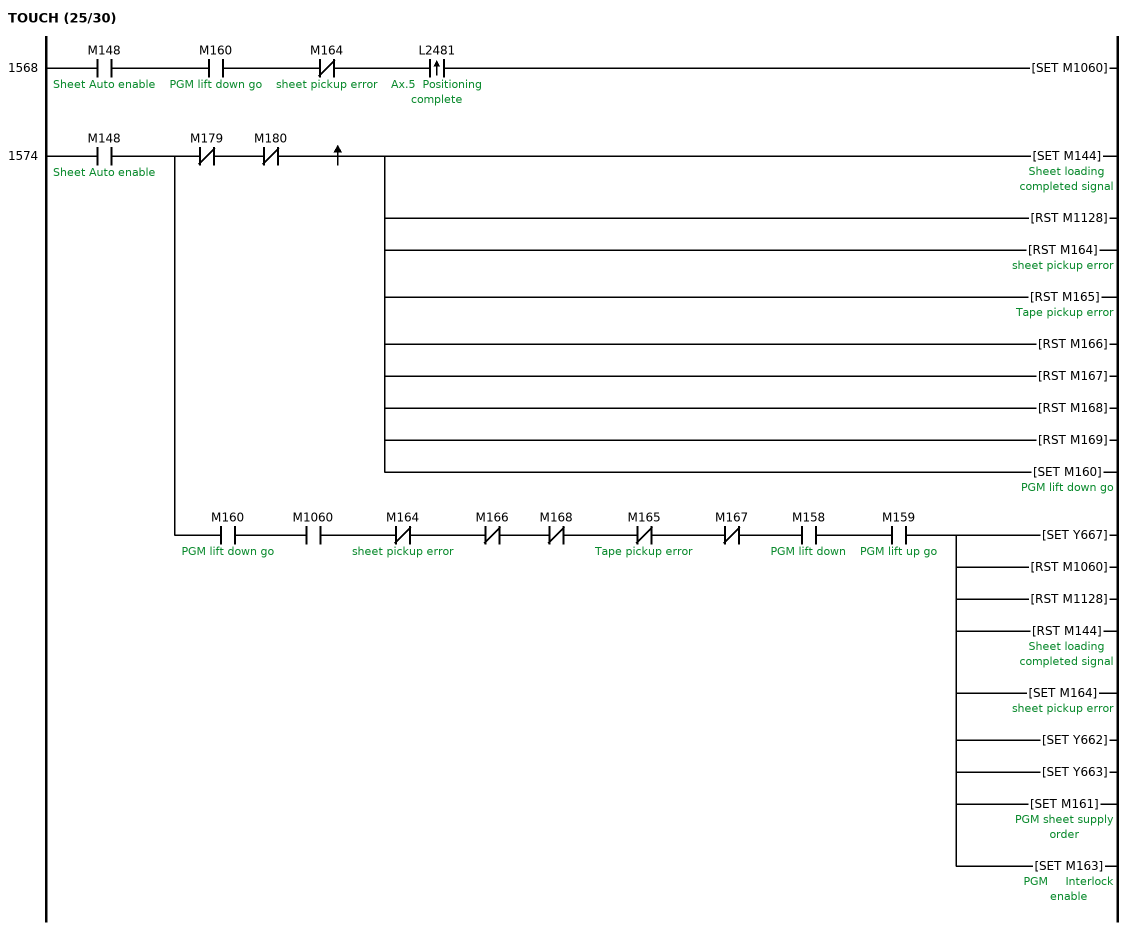
[picture p72: ladder of TOUCH, rungs at steps 1568 to 1574]
1568  LD      M148  ; Sheet Auto enable
      AND     M160  ; PGM lift down go
      ANI     M164  ; sheet pickup error
      ANDP    L2481  ; Ax.5  Positioning complete
      SET     M1060
1574  LD      M148  ; Sheet Auto enable
      MPS
      ANI     M179
      ANI     M180
      MEP
      SET     M144  ; Sheet loading completed signal
      RST     M1128
      RST     M164  ; sheet pickup error
      RST     M165  ; Tape pickup error
      RST     M166
      RST     M167
      RST     M168
      RST     M169
      SET     M160  ; PGM lift down go
      MPP
      AND     M160  ; PGM lift down go
      AND     M1060
      ANI     M164  ; sheet pickup error
      ANI     M166
      ANI     M168
      ANI     M165  ; Tape pickup error
      ANI     M167
      AND     M158  ; PGM lift down
      AND     M159  ; PGM lift up go
      SET     Y667
      RST     M1060
      RST     M1128
      RST     M144  ; Sheet loading completed signal
      SET     M164  ; sheet pickup error
      SET     Y662
      SET     Y663
      SET     M161  ; PGM sheet supply order
      SET     M163  ; PGM     Interlock enable
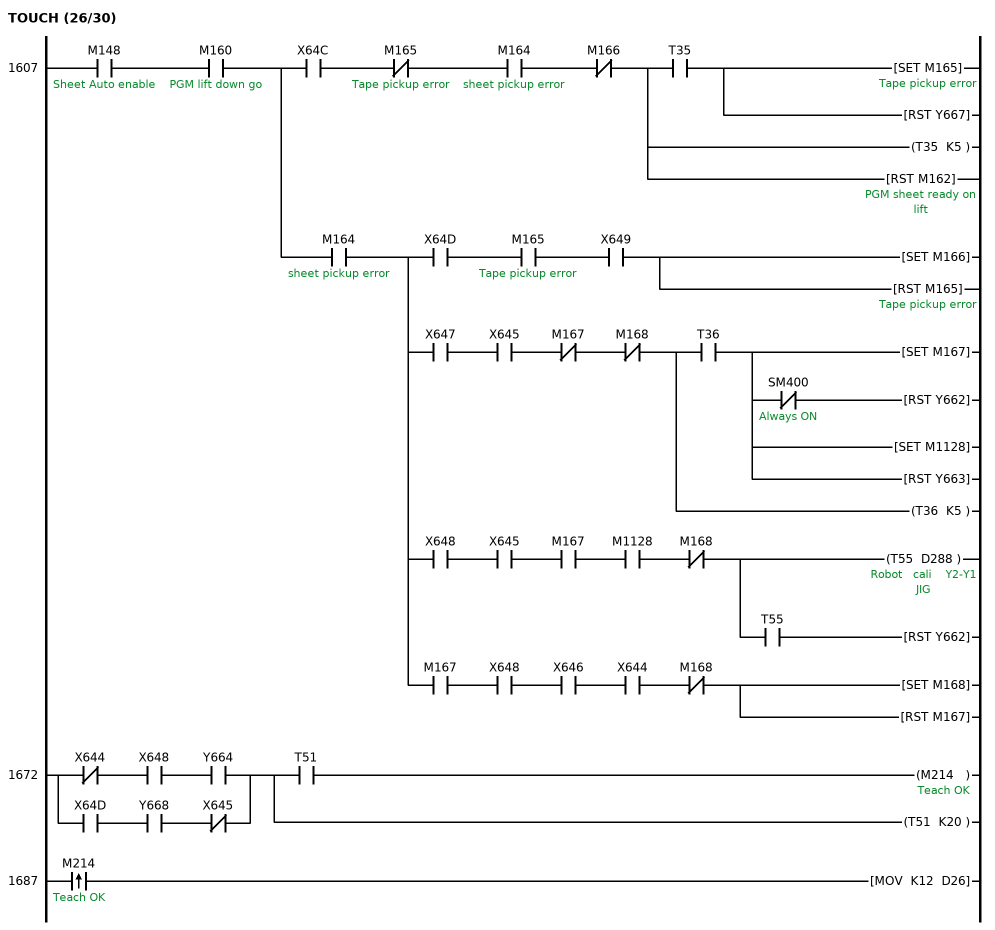
1607  LD      M148  ; Sheet Auto enable
      AND     M160  ; PGM lift down go
      MPS
      AND     X64C
      ANI     M165  ; Tape pickup error
      AND     M164  ; sheet pickup error
      ANI     M166
      MPS
      AND     T35
      SET     M165  ; Tape pickup error
      RST     Y667
      MPP
      OUT     T35 K5
      RST     M162  ; PGM sheet ready on lift
      MPP
      AND     M164  ; sheet pickup error
      MPS
      AND     X64D
      AND     M165  ; Tape pickup error
      AND     X649
      SET     M166
      RST     M165  ; Tape pickup error
      MRD
      AND     X647
      AND     X645
      ANI     M167
      ANI     M168
      MPS
      AND     T36
      SET     M167
      MPS
      ANI     SM400  ; Always ON
      RST     Y662
      MPP
      SET     M1128
      RST     Y663
      MPP
      OUT     T36 K5
      MRD
      AND     X648
      AND     X645
      AND     M167
      AND     M1128
      ANI     M168
      OUT     T55 D288  ; Robot   cali    Y2-Y1   JIG
      AND     T55
      RST     Y662
      MPP
      AND     M167
      AND     X648
      AND     X646
      AND     X644
      ANI     M168
      SET     M168
      RST     M167
1672  LDI     X644
      AND     X648
      AND     Y664
      LD      X64D
      AND     Y668
      ANI     X645
      ORB
      MPS
      AND     T51
      OUT     M214  ; Teach OK
      MPP
      OUT     T51 K20
1687  LDP     M214  ; Teach OK
      MOV     K12 D26
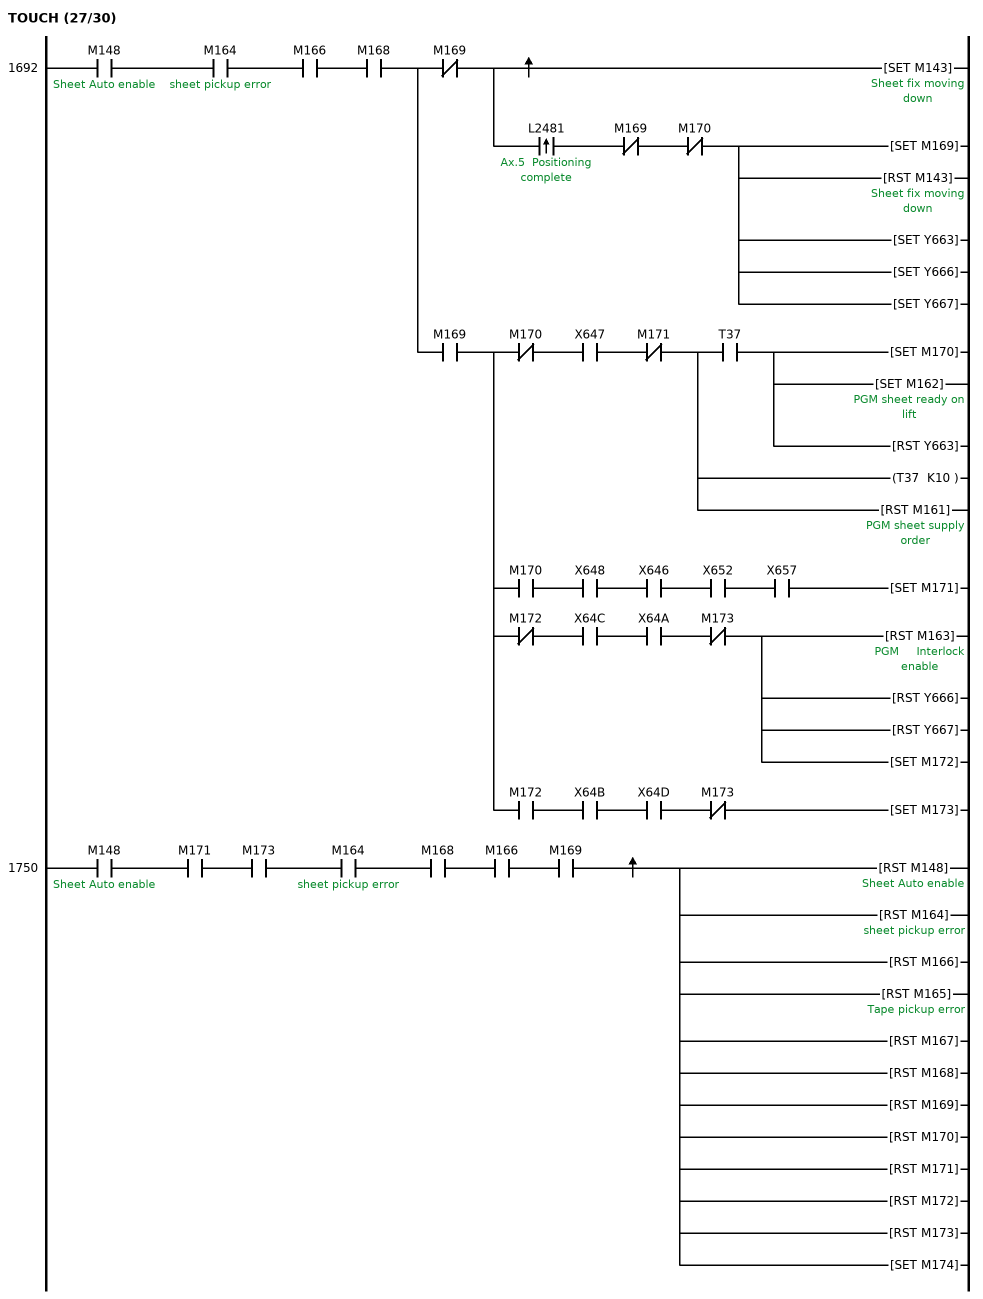
1692  LD      M148  ; Sheet Auto enable
      AND     M164  ; sheet pickup error
      AND     M166
      AND     M168
      MPS
      ANI     M169
      MPS
      MEP
      SET     M143  ; Sheet fix moving down
      MPP
      ANDP    L2481  ; Ax.5  Positioning complete
      ANI     M169
      ANI     M170
      SET     M169
      RST     M143  ; Sheet fix moving down
      SET     Y663
      SET     Y666
      SET     Y667
      MPP
      AND     M169
      MPS
      ANI     M170
      AND     X647
      ANI     M171
      MPS
      AND     T37
      SET     M170
      SET     M162  ; PGM sheet ready on lift
      RST     Y663
      MPP
      OUT     T37 K10
      RST     M161  ; PGM sheet supply order
      MRD
      AND     M170
      AND     X648
      AND     X646
      AND     X652
      AND     X657
      SET     M171
      MRD
      ANI     M172
      AND     X64C
      AND     X64A
      ANI     M173
      RST     M163  ; PGM     Interlock enable
      RST     Y666
      RST     Y667
      SET     M172
      MPP
      AND     M172
      AND     X64B
      AND     X64D
      ANI     M173
      SET     M173
1750  LD      M148  ; Sheet Auto enable
      AND     M171
      AND     M173
      AND     M164  ; sheet pickup error
      AND     M168
      AND     M166
      AND     M169
      MEP
      RST     M148  ; Sheet Auto enable
      RST     M164  ; sheet pickup error
      RST     M166
      RST     M165  ; Tape pickup error
      RST     M167
      RST     M168
      RST     M169
      RST     M170
      RST     M171
      RST     M172
      RST     M173
      SET     M174
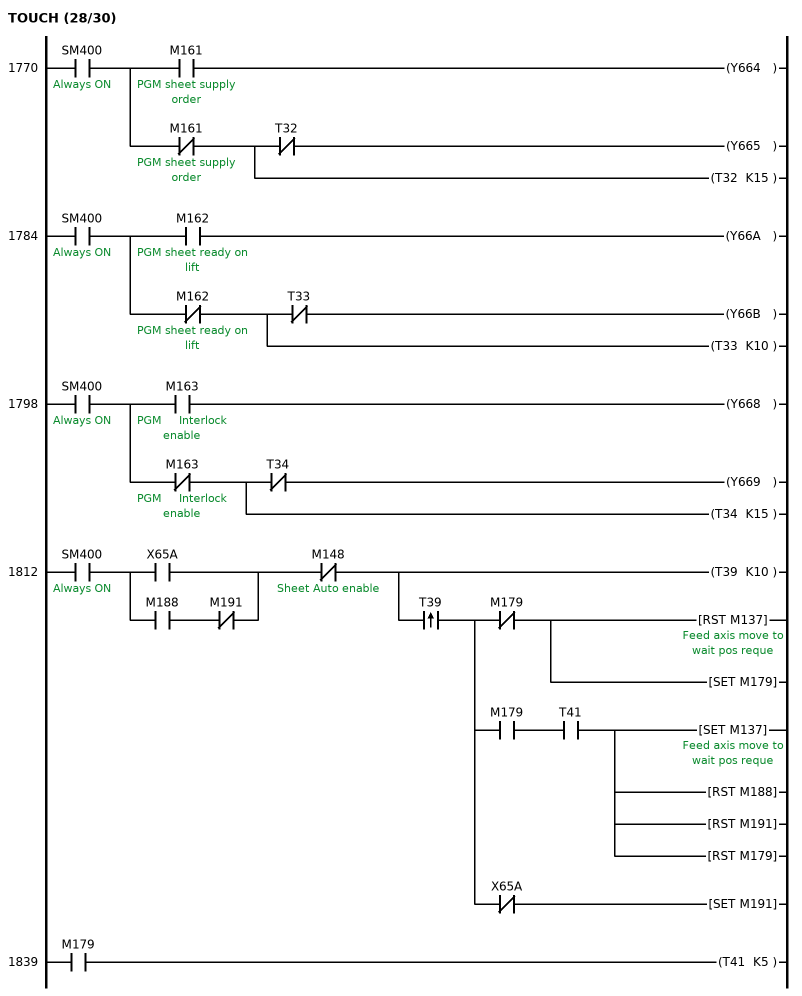
1770  LD      SM400  ; Always ON
      MPS
      AND     M161  ; PGM sheet supply order
      OUT     Y664
      MPP
      ANI     M161  ; PGM sheet supply order
      MPS
      ANI     T32
      OUT     Y665
      MPP
      OUT     T32 K15
1784  LD      SM400  ; Always ON
      MPS
      AND     M162  ; PGM sheet ready on lift
      OUT     Y66A
      MPP
      ANI     M162  ; PGM sheet ready on lift
      MPS
      ANI     T33
      OUT     Y66B
      MPP
      OUT     T33 K10
1798  LD      SM400  ; Always ON
      MPS
      AND     M163  ; PGM     Interlock enable
      OUT     Y668
      MPP
      ANI     M163  ; PGM     Interlock enable
      MPS
      ANI     T34
      OUT     Y669
      MPP
      OUT     T34 K15
1812  LD      SM400  ; Always ON
      LD      X65A
      LD      M188
      ANI     M191
      ORB
      ANB
      ANI     M148  ; Sheet Auto enable
      OUT     T39 K10
      ANDP    T39
      MPS
      ANI     M179
      RST     M137  ; Feed axis move to wait pos reque
      SET     M179
      MRD
      AND     M179
      AND     T41
      SET     M137  ; Feed axis move to wait pos reque
      RST     M188
      RST     M191
      RST     M179
      MPP
      ANI     X65A
      SET     M191
1839  LD      M179
      OUT     T41 K5
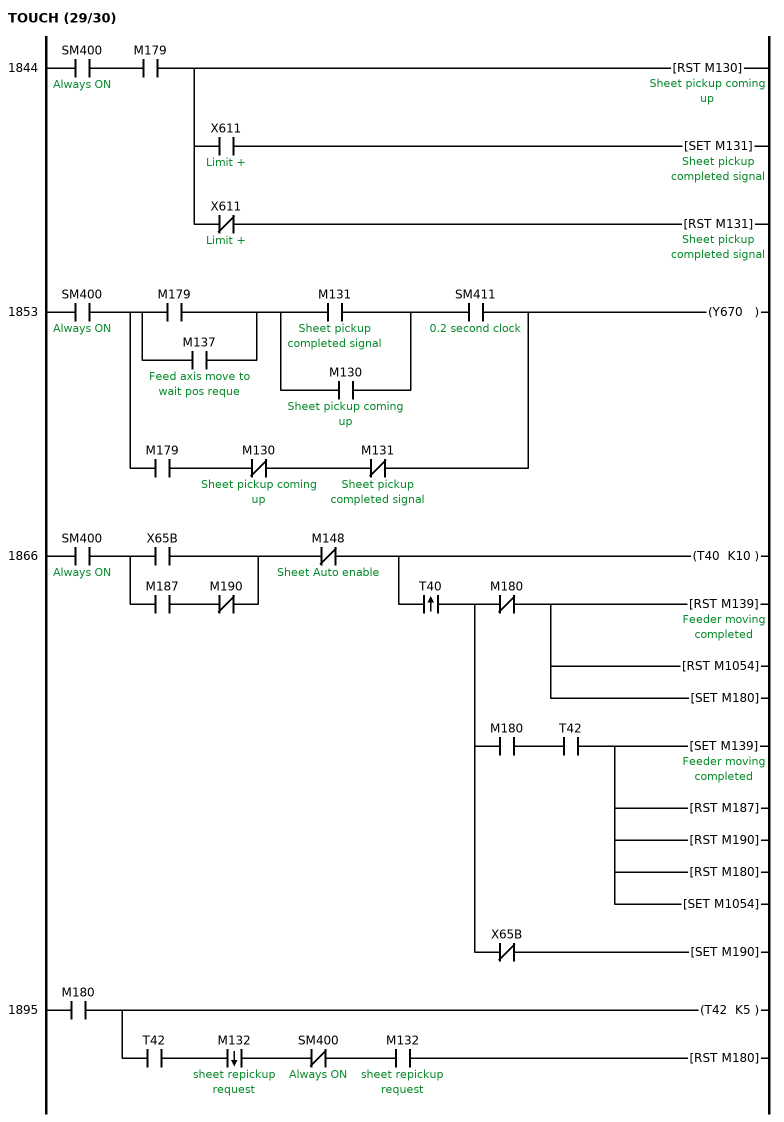
1844  LD      SM400  ; Always ON
      AND     M179
      RST     M130  ; Sheet pickup coming up
      MPS
      AND     X611  ; Limit +
      SET     M131  ; Sheet pickup completed signal
      MPP
      ANI     X611  ; Limit +
      RST     M131  ; Sheet pickup completed signal
1853  LD      SM400  ; Always ON
      LD      M179
      OR      M137  ; Feed axis move to wait pos reque
      LD      M131  ; Sheet pickup completed signal
      OR      M130  ; Sheet pickup coming up
      ANB
      AND     SM411  ; 0.2 second clock
      LD      M179
      ANI     M130  ; Sheet pickup coming up
      ANI     M131  ; Sheet pickup completed signal
      ORB
      ANB
      OUT     Y670
1866  LD      SM400  ; Always ON
      LD      X65B
      LD      M187
      ANI     M190
      ORB
      ANB
      ANI     M148  ; Sheet Auto enable
      OUT     T40 K10
      ANDP    T40
      MPS
      ANI     M180
      RST     M139  ; Feeder moving completed
      RST     M1054
      SET     M180
      MRD
      AND     M180
      AND     T42
      SET     M139  ; Feeder moving completed
      RST     M187
      RST     M190
      RST     M180
      SET     M1054
      MPP
      ANI     X65B
      SET     M190
1895  LD      M180
      OUT     T42 K5
      AND     T42
      ANDF    M132  ; sheet repickup request
      ANI     SM400  ; Always ON
      AND     M132  ; sheet repickup request
      RST     M180
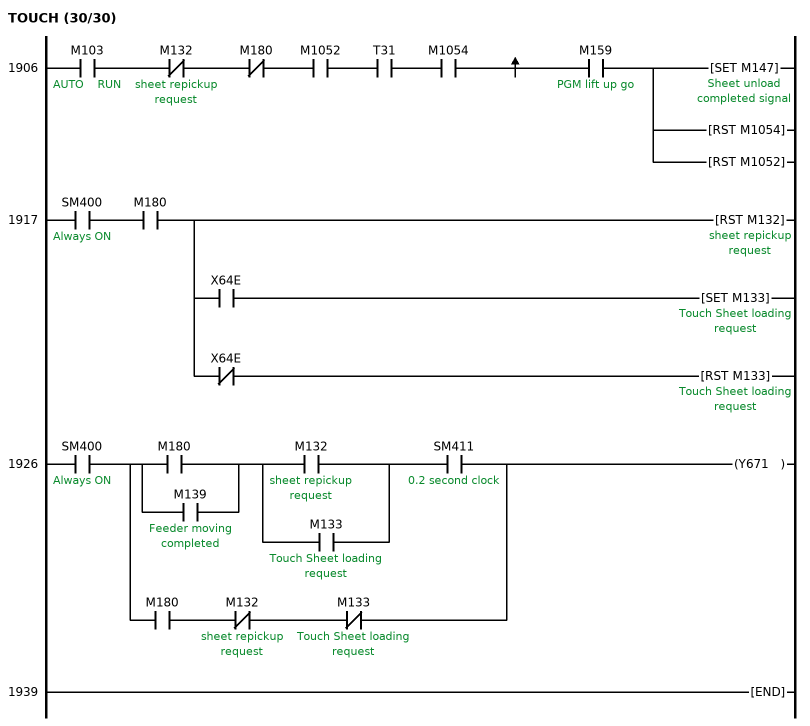
1906  LD      M103  ; AUTO    RUN
      ANI     M132  ; sheet repickup request
      ANI     M180
      AND     M1052
      AND     T31
      AND     M1054
      MEP
      AND     M159  ; PGM lift up go
      SET     M147  ; Sheet unload completed signal
      RST     M1054
      RST     M1052
1917  LD      SM400  ; Always ON
      AND     M180
      RST     M132  ; sheet repickup request
      MPS
      AND     X64E
      SET     M133  ; Touch Sheet loading request
      MPP
      ANI     X64E
      RST     M133  ; Touch Sheet loading request
1926  LD      SM400  ; Always ON
      LD      M180
      OR      M139  ; Feeder moving completed
      LD      M132  ; sheet repickup request
      OR      M133  ; Touch Sheet loading request
      ANB
      AND     SM411  ; 0.2 second clock
      LD      M180
      ANI     M132  ; sheet repickup request
      ANI     M133  ; Touch Sheet loading request
      ORB
      ANB
      OUT     Y671
1939  END
END_PROGRAM

PROGRAM VISION
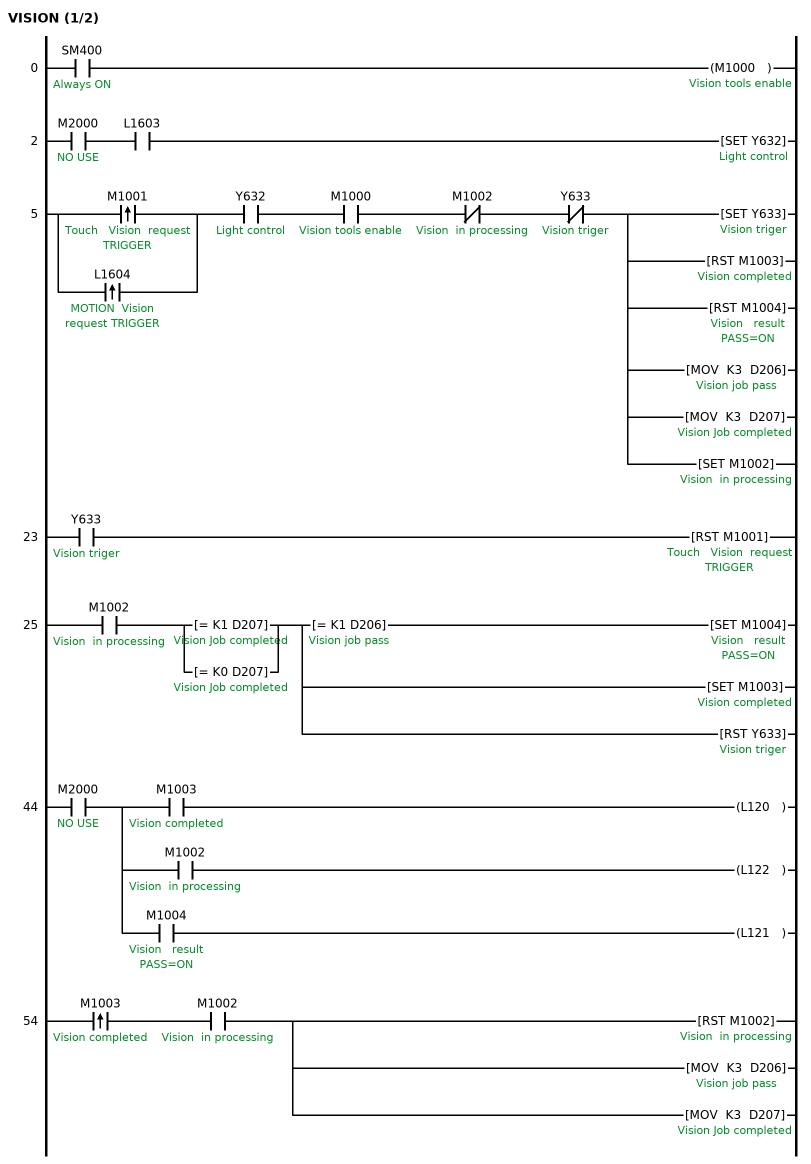
0     LD      SM400  ; Always ON
      OUT     M1000  ; Vision tools enable
2     LD      M2000  ; NO USE
      AND     L1603
      SET     Y632  ; Light control
5     LDP     M1001  ; Touch   Vision  request TRIGGER
      ORP     L1604  ; MOTION  Vision  request TRIGGER
      AND     Y632  ; Light control
      AND     M1000  ; Vision tools enable
      ANI     M1002  ; Vision  in processing
      ANI     Y633  ; Vision triger
      SET     Y633  ; Vision triger
      RST     M1003  ; Vision completed
      RST     M1004  ; Vision   result PASS=ON
      MOV     K3 D206  ; Vision job pass
      MOV     K3 D207  ; Vision Job completed
      SET     M1002  ; Vision  in processing
23    LD      Y633  ; Vision triger
      RST     M1001  ; Touch   Vision  request TRIGGER
25    LD      M1002  ; Vision  in processing
      LD=     K1 D207  ; Vision Job completed
      OR=     K0 D207  ; Vision Job completed
      ANB
      MPS
      AND=    K1 D206  ; Vision job pass
      SET     M1004  ; Vision   result PASS=ON
      MPP
      SET     M1003  ; Vision completed
      RST     Y633  ; Vision triger
44    LD      M2000  ; NO USE
      MPS
      AND     M1003  ; Vision completed
      OUT     L120
      MRD
      AND     M1002  ; Vision  in processing
      OUT     L122
      MPP
      AND     M1004  ; Vision   result PASS=ON
      OUT     L121
54    LDP     M1003  ; Vision completed
      AND     M1002  ; Vision  in processing
      RST     M1002  ; Vision  in processing
      MOV     K3 D206
      MOV     K3 D207
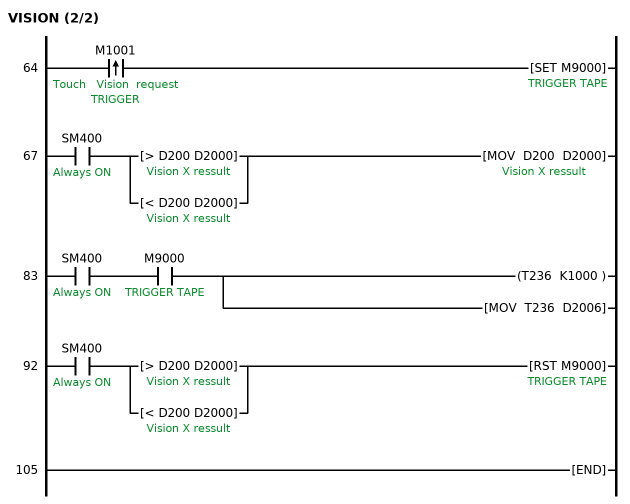
64    LDP     M1001  ; Touch   Vision  request TRIGGER
      SET     M9000  ; TRIGGER TAPE
67    LD      SM400  ; Always ON
      LD>     D200 D2000  ; Vision X ressult
      OR<     D200 D2000  ; Vision X ressult
      ANB
      MOV     D200 D2000
83    LD      SM400  ; Always ON
      AND     M9000  ; TRIGGER TAPE
      OUT     T236 K1000
      MOV     T236 D2006
92    LD      SM400  ; Always ON
      LD>     D200 D2000  ; Vision X ressult
      OR<     D200 D2000  ; Vision X ressult
      ANB
      RST     M9000  ; TRIGGER TAPE
105   END
END_PROGRAM

// device comments not shown above
X608  ; Vaccum pressure signal
X609  ; Change Tape
X61A  ; Fix sheet cylinder pos
X61E  ; Up Position
M10  ; Head Select
M30  ; Jig Vacuum-Blow
M219  ; CALIB OK
M220  ; CALIB   JIG OK
M270  ; SP_TRIG MCR
M300  ; nâng hạ bàn đặt Tape
M500  ; PROCESS PASS
M501  ; 1: DÁN 0: BỎ  QUA
M505  ; LUÔN   DÁN    TAPE
M1015  ; Vision  result  PASS=ON JIG1
M1024  ; Vision  result  PASS=ON JIG2
M1042  ; Get     vision  master  JIG
M1065  ; Robot   calib   Pos 1   get JIG
M1066  ; Robot   calib   Pos 2   get JIG
M1067  ; Robot   calib   excute  JIG
M1193  ; NO USE
D18  ; Sheet Rows
D20  ; Sheet rows index
D22  ; sheet repickup counter
D50  ; Vision X ressult JIG 1
D52  ; Vision Y result JIG 1
D54  ; Vision  angle JIG 1
D70  ; Vision X ressult JIG 2
D72  ; Vision Y result JIG 2
D74  ; Vision  angle JIG 2
D240  ; RB-CAM  RATE X  JIG
D242  ; RB-CAM  RATE Y  JIG
D250  ; Vision master X JIG1
D252  ; Vision master Y JIG1
D254  ; Vision master Angle JIG1
D260  ; Vision master X JIG2
D262  ; Vision master Y JIG2
D264  ; Vision master Angle JIG2
D270  ; Robot   cali X1 JIG
D272  ; Robot   cali Y1 JIG
D274  ; Robot   cali XC1 JIG
D276  ; Robot   cali YC1 JIG
D278  ; Robot   cali    X2-X1   JIG
D280  ; Robot   cali X2 JIG
D282  ; Robot   cali Y2 JIG
D286  ; Robot   cali YC2 JIG
D302  ; DO LECH YC JIG1
D304  ; GOCS2-  GÓC1   JIG1
D306  ; DO LECH XC JIG2
D308  ; DO LECH YC JIG2
D310  ; GOCS2-  GÓC1   JIG2    FLOAD
D312  ; BÙ XUNG XC JIG1
D314  ; BÙ XUNG YC JIG1
D316  ; BÙ XUNG XC JIG2
D318  ; BÙ XUNG YC JIG2
D320  ; INT BÙ XUNG JIG1 XC
D322  ; INT BÙ XUNG JIG1 YC
D380  ; VISION  HEAD 1  ANGLE
D382  ; VISION  HEAD 2  ANGLE
D48008  ; SPEED Z1 MANUAL
D48018  ; SPEED R1 MANUAL
D48028  ; SPEED Z2 MANUAL
D48038  ; SPEED R2 MANUAL
D48048  ; SPEED F MANUAL
D48050  ; ADRES X
D48052  ; SPEED X
D48058  ; SPEED X MANUAL
D48060  ; ADRES Y
D48062  ; SPEED Y
D48068  ; SPEED Y MANUAL
D48120  ; TIME    DELAY   RUN Z1, R1
D48640  ; Ax.1 JOG speed setting
D48641  ; Ax.1 JOG speed setting
D48642  ; Ax.2 JOG speed setting
D48643  ; Ax.2 JOG speed setting
D48644  ; Ax.3 JOG speed setting
D48645  ; Ax.3 JOG speed setting
D48646  ; Ax.4 JOG speed setting
D48647  ; Ax.4 JOG speed setting
D48648  ; Ax.5 JOG speed setting
D48649  ; Ax.5 JOG speed setting
D48650  ; Ax.6 JOG speed setting
D48651  ; Ax.6 JOG speed setting
D48652  ; Ax.7 JOG speed setting
D48653  ; Ax.7 JOG speed setting
D48654  ; Ax.8 JOG speed setting
D48655  ; Ax.8 JOG speed setting
D49000  ; Ax.1  Feed current value/Roller
D49001  ; Ax.1  Feed current value/Roller
D49003  ; Ax.1  Real current value
D49004  ; Ax.1  Deviation counter value
D49005  ; Ax.1  Deviation counter value
D49006  ; Ax.1  Minor error code
D49007  ; Ax.1  Major error code
D49008  ; Ax.1  Servo error code
D49009  ; Ax.1  Home position return re-mo
D49010  ; Ax.1  Movement amount after prox
D49011  ; Ax.1  Movement amount after prox
D49012  ; Ax.1  Execute program No.
D49013  ; Ax.1 M-code
D49014  ; Ax.1  Torque limit value
D49015  ; Ax.1  Data set pointer for const
D49018  ; Ax.1  Real current value at stop
D49019  ; Ax.1  Real current value at stop
D49020  ; Ax.2  Feed current value/Roller
D49021  ; Ax.2  Feed current value/Roller
D49023  ; Ax.2  Real current value
D49024  ; Ax.2  Deviation counter value
D49025  ; Ax.2  Deviation counter value
D49026  ; Ax.2  Minor error code
D49027  ; Ax.2  Major error code
D49028  ; Ax.2  Servo error code
D49029  ; Ax.2  Home position return re-mo
D49030  ; Ax.2  Movement amount after prox
D49031  ; Ax.2  Movement amount after prox
D49032  ; Ax.2  Execute program No.
D49033  ; Ax.2 M-code
D49034  ; Ax.2  Torque limit value
D49035  ; Ax.2  Data set pointer for const
D49038  ; Ax.2  Real current value at stop
D49039  ; Ax.2  Real current value at stop
D49040  ; Ax.3  Feed current value/Roller
D49041  ; Ax.3  Feed current value/Roller
D49043  ; Ax.3  Real current value
D49044  ; Ax.3  Deviation counter value
D49045  ; Ax.3  Deviation counter value
D49046  ; Ax.3  Minor error code
D49047  ; Ax.3  Major error code
D49048  ; Ax.3  Servo error code
D49049  ; Ax.3  Home position return re-mo
D49050  ; Ax.3  Movement amount after prox
D49051  ; Ax.3  Movement amount after prox
D49052  ; Ax.3  Execute program No.
D49053  ; Ax.3 M-code
D49054  ; Ax.3  Torque limit value
D49055  ; Ax.3  Data set pointer for const
D49058  ; Ax.3  Real current value at stop
D49059  ; Ax.3  Real current value at stop
D49060  ; Ax.4  Feed current value/Roller
D49061  ; Ax.4  Feed current value/Roller
D49063  ; Ax.4  Real current value
D49064  ; Ax.4  Deviation counter value
D49065  ; Ax.4  Deviation counter value
D49066  ; Ax.4  Minor error code
D49067  ; Ax.4  Major error code
D49068  ; Ax.4  Servo error code
D49069  ; Ax.4  Home position return re-mo
D49070  ; Ax.4  Movement amount after prox
D49071  ; Ax.4  Movement amount after prox
D49072  ; Ax.4  Execute program No.
D49073  ; Ax.4 M-code
D49074  ; Ax.4  Torque limit value
D49075  ; Ax.4  Data set pointer for const
D49078  ; Ax.4  Real current value at stop
D49079  ; Ax.4  Real current value at stop
D49080  ; Ax.5  Feed current value/Roller
D49081  ; Ax.5  Feed current value/Roller
D49083  ; Ax.5  Real current value
D49084  ; Ax.5  Deviation counter value
D49085  ; Ax.5  Deviation counter value
D49086  ; Ax.5  Minor error code
D49087  ; Ax.5  Major error code
D49088  ; Ax.5  Servo error code
D49089  ; Ax.5  Home position return re-mo
D49090  ; Ax.5  Movement amount after prox
D49091  ; Ax.5  Movement amount after prox
D49092  ; Ax.5  Execute program No.
D49093  ; Ax.5 M-code
D49094  ; Ax.5  Torque limit value
D49095  ; Ax.5  Data set pointer for const
D49098  ; Ax.5  Real current value at stop
D49099  ; Ax.5  Real current value at stop
D49100  ; Ax.6  Feed current value/Roller
D49101  ; Ax.6  Feed current value/Roller
D49103  ; Ax.6  Real current value
D49104  ; Ax.6  Deviation counter value
D49105  ; Ax.6  Deviation counter value
D49106  ; Ax.6  Minor error code
D49107  ; Ax.6  Major error code
D49108  ; Ax.6  Servo error code
D49109  ; Ax.6  Home position return re-mo
D49110  ; Ax.6  Movement amount after prox
D49111  ; Ax.6  Movement amount after prox
D49112  ; Ax.6  Execute program No.
D49113  ; Ax.6 M-code
D49114  ; Ax.6  Torque limit value
D49115  ; Ax.6  Data set pointer for const
D49118  ; Ax.6  Real current value at stop
D49119  ; Ax.6  Real current value at stop
D49120  ; Ax.7  Feed current value/Roller
D49121  ; Ax.7  Feed current value/Roller
D49123  ; Ax.7  Real current value
D49124  ; Ax.7  Deviation counter value
D49125  ; Ax.7  Deviation counter value
D49126  ; Ax.7  Minor error code
D49127  ; Ax.7  Major error code
D49128  ; Ax.7  Servo error code
D49129  ; Ax.7  Home position return re-mo
D49130  ; Ax.7  Movement amount after prox
D49131  ; Ax.7  Movement amount after prox
D49132  ; Ax.7  Execute program No.
D49133  ; Ax.7 M-code
D49134  ; Ax.7  Torque limit value
D49135  ; Ax.7  Data set pointer for const
D49138  ; Ax.7  Real current value at stop
D49139  ; Ax.7  Real current value at stop
D49140  ; Ax.8  Feed current value/Roller
D49141  ; Ax.8  Feed current value/Roller
D49142  ; Ax.8  Real current value
D49143  ; Ax.8  Real current value
D49144  ; Ax.8  Deviation counter value
D49145  ; Ax.8  Deviation counter value
D49146  ; Ax.8  Minor error code
D49147  ; Ax.8  Major error code
D49148  ; Ax.8  Servo error code
D49149  ; Ax.8  Home position return re-mo
D49150  ; Ax.8  Movement amount after prox
D49151  ; Ax.8  Movement amount after prox
D49152  ; Ax.8  Execute program No.
D49153  ; Ax.8 M-code
D49154  ; Ax.8  Torque limit value
D49155  ; Ax.8  Data set pointer for const
D49158  ; Ax.8  Real current value at stop
D49159  ; Ax.8  Real current value at stop
D49704  ; PLC ready flag request
D49705  ; Speed switching point specified
D49706  ; All axes servo ON command reques
D49714  ; Manual pulse generator 1 axis No
D49715  ; Manual pulse generator 1 axis No
D49716  ; Manual pulse generator 2 axis No
D49717  ; Manual pulse generator 2 axis No
D49718  ; Manual pulse generator 3 axis No
D49719  ; Manual pulse generator 3 axis No
D49720  ; Ax.1  ManualPulseGen. 1Pls. inpu
D49721  ; Ax.2  ManualPulseGen. 1Pls. inpu
D49722  ; Ax.3  ManualPulseGen. 1Pls. inpu
D49723  ; Ax.4  ManualPulseGen. 1Pls. inpu
D49724  ; Ax.5  ManualPulseGen. 1Pls. inpu
D49725  ; Ax.6  ManualPulseGen. 1Pls. inpu
D49726  ; Ax.7  ManualPulseGen. 1Pls. inpu
D49727  ; Ax.8  ManualPulseGen. 1Pls. inpu
D49752  ; Manual pulse generator 1 smoothi
D49753  ; Manual pulse generator 2 smoothi
D49754  ; Manual pulse generator 3 smoothi
D49755  ; Manual pulse generator 1 enable
D49756  ; Manual pulse generator 2 enable
D49757  ; Manual pulse generator 3 enable
D49800  ; Virtual servo  Ax.1  Feed curren
D49801  ; Virtual servo  Ax.1  Feed curren
D49802  ; Virtual servo  Ax.1  Minor error
D49803  ; Virtual servo  Ax.1  Major error
D49804  ; Virtual servo  Ax.1  Execute pro
D49805  ; Virtual servo  Ax.1  M-code
D49806  ; Virtual servo  Ax.1  Current val
D49807  ; Virtual servo  Ax.1  Current val
D49808  ; Virtual servo  Ax.1  Error searc
D49809  ; Virtual servo  Ax.1  Data set po
D49810  ; Virtual servo  Ax.2  Feed curren
D49811  ; Virtual servo  Ax.2  Feed curren
D49812  ; Virtual servo  Ax.2  Minor error
D49813  ; Virtual servo  Ax.2  Major error
D49814  ; Virtual servo  Ax.2  Execute pro
D49815  ; Virtual servo  Ax.2  M-code
D49816  ; Virtual servo  Ax.2  Current val
D49817  ; Virtual servo  Ax.2  Current val
D49818  ; Virtual servo  Ax.2  Error searc
D49819  ; Virtual servo  Ax.2  Data set po
D49820  ; Virtual servo  Ax.3  Feed curren
D49821  ; Virtual servo  Ax.3  Feed curren
D49822  ; Virtual servo  Ax.3  Minor error
D49823  ; Virtual servo  Ax.3  Major error
D49824  ; Virtual servo  Ax.3  Execute pro
D49825  ; Virtual servo  Ax.3  M-code
D49826  ; Virtual servo  Ax.3  Current val
D49827  ; Virtual servo  Ax.3  Current val
D49828  ; Virtual servo  Ax.3  Error searc
D49829  ; Virtual servo  Ax.3  Data set po
D49830  ; Virtual servo  Ax.4  Feed curren
D49831  ; Virtual servo  Ax.4  Feed curren
D49832  ; Virtual servo  Ax.4  Minor error
D49833  ; Virtual servo  Ax.4  Major error
D49834  ; Virtual servo  Ax.4  Execute pro
D49835  ; Virtual servo  Ax.4  M-code
D49836  ; Virtual servo  Ax.4  Current val
D49837  ; Virtual servo  Ax.4  Current val
D49838  ; Virtual servo  Ax.4  Error searc
D49839  ; Virtual servo  Ax.4  Data set po
D49840  ; Virtual servo  Ax.5  Feed curren
D49841  ; Virtual servo  Ax.5  Feed curren
D49842  ; Virtual servo  Ax.5  Minor error
D49843  ; Virtual servo  Ax.5  Major error
D49844  ; Virtual servo  Ax.5  Execute pro
D49845  ; Virtual servo  Ax.5  M-code
D49846  ; Virtual servo  Ax.5  Current val
D49847  ; Virtual servo  Ax.5  Current val
D49848  ; Virtual servo  Ax.5  Error searc
D49849  ; Virtual servo  Ax.5  Data set po
D49850  ; Virtual servo  Ax.6  Feed curren
D49851  ; Virtual servo  Ax.6  Feed curren
D49852  ; Virtual servo  Ax.6  Minor error
D49853  ; Virtual servo  Ax.6  Major error
D49854  ; Virtual servo  Ax.6  Execute pro
D49855  ; Virtual servo  Ax.6  M-code
D49856  ; Virtual servo  Ax.6  Current val
D49857  ; Virtual servo  Ax.6  Current val
D49858  ; Virtual servo  Ax.6  Error searc
D49859  ; Virtual servo  Ax.6  Data set po
D49860  ; Virtual servo  Ax.7  Feed curren
D49861  ; Virtual servo  Ax.7  Feed curren
D49862  ; Virtual servo  Ax.7  Minor error
D49863  ; Virtual servo  Ax.7  Major error
D49864  ; Virtual servo  Ax.7  Execute pro
D49865  ; Virtual servo  Ax.7  M-code
D49866  ; Virtual servo  Ax.7  Current val
D49867  ; Virtual servo  Ax.7  Current val
D49868  ; Virtual servo  Ax.7  Error searc
D49869  ; Virtual servo  Ax.7  Data set po
D49870  ; Virtual servo  Ax.8  Feed curren
D49871  ; Virtual servo  Ax.8  Feed curren
D49872  ; Virtual servo  Ax.8  Minor error
D49873  ; Virtual servo  Ax.8  Major error
D49874  ; Virtual servo  Ax.8  Execute pro
D49875  ; Virtual servo  Ax.8  M-code
D49876  ; Virtual servo  Ax.8  Current val
D49877  ; Virtual servo  Ax.8  Current val
D49878  ; Virtual servo  Ax.8  Error searc
D49879  ; Virtual servo  Ax.8  Data set po
D50122  ; Sync. encoder  Ax.1  Minor error
D50123  ; Sync. encoder  Ax.1  Major error
D50128  ; Sync. encoder  Ax.1  Error searc
D50132  ; Sync. encoder  Ax.2  Minor error
D50133  ; Sync. encoder  Ax.2  Major error
D50138  ; Sync. encoder  Ax.2  Error searc
D50142  ; Sync. encoder  Ax.3  Minor error
D50143  ; Sync. encoder  Ax.3  Major error
D50148  ; Sync. encoder  Ax.3  Error searc
D50152  ; Sync. encoder  Ax.4  Minor error
D50153  ; Sync. encoder  Ax.4  Major error
D50158  ; Sync. encoder  Ax.4  Error searc
D50162  ; Sync. encoder  Ax.5  Minor error
D50163  ; Sync. encoder  Ax.5  Major error
D50168  ; Sync. encoder  Ax.5  Error searc
D50172  ; Sync. encoder  Ax.6  Minor error
D50173  ; Sync. encoder  Ax.6  Major error
D50178  ; Sync. encoder  Ax.6  Error searc
D50182  ; Sync. encoder  Ax.7  Minor error
D50183  ; Sync. encoder  Ax.7  Major error
D50188  ; Sync. encoder  Ax.7  Error searc
D50192  ; Sync. encoder  Ax.8  Minor error
D50193  ; Sync. encoder  Ax.8  Major error
D50198  ; Sync. encoder  Ax.8  Error searc
D50241  ; Cam  Ax.1  Execute cam No.
D50242  ; Cam  Ax.1  Execute stroke amount
D50243  ; Cam  Ax.1  Execute stroke amount
D50244  ; Cam  Ax.1  Cam axis current valu
D50245  ; Cam  Ax.1  Cam axis current valu
D50251  ; Cam  Ax.2  Execute cam No.
D50252  ; Cam  Ax.2  Execute stroke amount
D50253  ; Cam  Ax.2  Execute stroke amount
D50254  ; Cam  Ax.2  Cam axis current valu
D50255  ; Cam  Ax.2  Cam axis current valu
D50261  ; Cam  Ax.3  Execute cam No.
D50262  ; Cam  Ax.3  Execute stroke amount
D50263  ; Cam  Ax.3  Execute stroke amount
D50264  ; Cam  Ax.3  Cam axis current valu
D50265  ; Cam  Ax.3  Cam axis current valu
D50271  ; Cam  Ax.4  Execute cam No.
D50272  ; Cam  Ax.4  Execute stroke amount
D50273  ; Cam  Ax.4  Execute stroke amount
D50274  ; Cam  Ax.4  Cam axis current valu
D50275  ; Cam  Ax.4  Cam axis current valu
D50281  ; Cam  Ax.5  Execute cam No.
D50282  ; Cam  Ax.5  Execute stroke amount
D50283  ; Cam  Ax.5  Execute stroke amount
D50284  ; Cam  Ax.5  Cam axis current valu
D50285  ; Cam  Ax.5  Cam axis current valu
D50291  ; Cam  Ax.6  Execute cam No.
D50292  ; Cam  Ax.6  Execute stroke amount
D50293  ; Cam  Ax.6  Execute stroke amount
D50294  ; Cam  Ax.6  Cam axis current valu
D50295  ; Cam  Ax.6  Cam axis current valu
D50301  ; Cam  Ax.7  Execute cam No.
D50302  ; Cam  Ax.7  Execute stroke amount
D50303  ; Cam  Ax.7  Execute stroke amount
D50304  ; Cam  Ax.7  Cam axis current valu
D50305  ; Cam  Ax.7  Cam axis current valu
D50311  ; Cam  Ax.8  Execute cam No.
D50312  ; Cam  Ax.8  Execute stroke amount
D50313  ; Cam  Ax.8  Execute stroke amount
D50314  ; Cam  Ax.8  Cam axis current valu
D50315  ; Cam  Ax.8  Cam axis current valu
Y623  ; Vaccum control
Y62B  ; Cylinder control
Y62C  ; Vaccum control
Y634  ; Vacum control
Y640  ; Light control
Y641  ; Vision triger
Y642  ; Light control
Y643  ; Vision triger
Y644  ; Change Tape
L2000  ; PLC ready flag
L2008  ; Ax.8  Start accept flag
L2035  ; Motion error history clear reque
L2038  ; Motion SFC debugging flag
L2039  ; Motion error detection flag
L2040  ; Speed switching point specified
L2041  ; System setting error flag
L2042  ; All axes servo ON command
L2046  ; Out-of-sync warning
L2047  ; Motion slot fault detection flag
L2049  ; All axes servo ON accept flag
L2051  ; Manual pulse generator 1 enable
L2052  ; Manual pulse generator 2 enable
L2053  ; Manual pulse generator 3 enable
L2054  ; Operation cycle over flag
L2061  ; Ax.1  Speed change accepting fla
L2062  ; Ax.2  Speed change accepting fla
L2063  ; Ax.3  Speed change accepting fla
L2064  ; Ax.4  Speed change accepting fla
L2065  ; Ax.5  Speed change accepting fla
L2066  ; Ax.6  Speed change accepting fla
L2067  ; Ax.7  Speed change accepting fla
L2068  ; Ax.8  Speed change accepting fla
L2101  ; Ax.1  Synchronous encoder curren
L2102  ; Ax.2  Synchronous encoder curren
L2103  ; Ax.3  Synchronous encoder curren
L2104  ; Ax.4  Synchronous encoder curren
L2105  ; Ax.5  Synchronous encoder curren
L2106  ; Ax.6  Synchronous encoder curren
L2107  ; Ax.7  Synchronous encoder curren
L2108  ; Ax.8  Synchronous encoder curren
L2128  ; Ax.1  Automatic decelerating fla
L2129  ; Ax.2  Automatic decelerating fla
L2130  ; Ax.3  Automatic decelerating fla
L2131  ; Ax.4  Automatic decelerating fla
L2132  ; Ax.5  Automatic decelerating fla
L2133  ; Ax.6  Automatic decelerating fla
L2134  ; Ax.7  Automatic decelerating fla
L2135  ; Ax.8  Automatic decelerating fla
L2240  ; Ax.1  Speed change "0" accepting
L2241  ; Ax.2  Speed change "0" accepting
L2242  ; Ax.3  Speed change "0" accepting
L2243  ; Ax.4  Speed change "0" accepting
L2244  ; Ax.5  Speed change "0" accepting
L2245  ; Ax.6  Speed change "0" accepting
L2246  ; Ax.7  Speed change "0" accepting
L2247  ; Ax.8  Speed change "0" accepting
L2272  ; Ax.1  Control loop monitor statu
L2273  ; Ax.2  Control loop monitor statu
L2274  ; Ax.3  Control loop monitor statu
L2275  ; Ax.4  Control loop monitor statu
L2276  ; Ax.5  Control loop monitor statu
L2277  ; Ax.6  Control loop monitor statu
L2278  ; Ax.7  Control loop monitor statu
L2279  ; Ax.8  Control loop monitor statu
L2400  ; Ax.1  Positioning start complete
L2402  ; Ax.1  In-position
L2403  ; Ax.1  Command in-position
L2404  ; Ax.1  Speed controlling
L2405  ; Ax.1  Speed-position switching l
L2406  ; Ax.1  Zero pass
L2409  ; Ax.1  Home position return reque
L2411  ; Ax.1  External signals FLS
L2412  ; Ax.1  External signals RLS
L2413  ; Ax.1  External signals STOP
L2414  ; Ax.1  External signals DOG/CHANG
L2415  ; Ax.1  Servo ready
L2416  ; Ax.1  Torque limiting
L2418  ; Ax.1  Virtual mode continuation
L2419  ; Ax.1 M-code outputting
L2420  ; Ax.2  Positioning start complete
L2422  ; Ax.2  In-position
L2423  ; Ax.2  Command in-position
L2424  ; Ax.2  Speed controlling
L2425  ; Ax.2  Speed-position switching l
L2426  ; Ax.2  Zero pass
L2429  ; Ax.2  Home position return reque
L2431  ; Ax.2  External signals FLS
L2432  ; Ax.2  External signals RLS
L2433  ; Ax.2  External signals STOP
L2434  ; Ax.2  External signals DOG/CHANG
L2435  ; Ax.2  Servo ready
L2436  ; Ax.2  Torque limiting
L2438  ; Ax.2  Virtual mode continuation
L2439  ; Ax.2 M-code outputting
L2440  ; Ax.3  Positioning start complete
L2442  ; Ax.3  In-position
L2443  ; Ax.3  Command in-position
L2444  ; Ax.3  Speed controlling
L2445  ; Ax.3  Speed-position switching l
L2446  ; Ax.3  Zero pass
L2449  ; Ax.3  Home position return reque
L2451  ; Ax.3  External signals FLS
L2452  ; Ax.3  External signals RLS
L2453  ; Ax.3  External signals STOP
L2454  ; Ax.3  External signals DOG/CHANG
L2455  ; Ax.3  Servo ready
L2456  ; Ax.3  Torque limiting
L2458  ; Ax.3  Virtual mode continuation
L2459  ; Ax.3 M-code outputting
L2460  ; Ax.4  Positioning start complete
L2462  ; Ax.4  In-position
L2463  ; Ax.4  Command in-position
L2464  ; Ax.4  Speed controlling
L2465  ; Ax.4  Speed-position switching l
L2466  ; Ax.4  Zero pass
L2469  ; Ax.4  Home position return reque
L2471  ; Ax.4  External signals FLS
L2472  ; Ax.4  External signals RLS
L2473  ; Ax.4  External signals STOP
L2474  ; Ax.4  External signals DOG/CHANG
L2475  ; Ax.4  Servo ready
L2476  ; Ax.4  Torque limiting
L2478  ; Ax.4  Virtual mode continuation
L2479  ; Ax.4 M-code outputting
L2480  ; Ax.5  Positioning start complete
L2482  ; Ax.5  In-position
L2483  ; Ax.5  Command in-position
L2484  ; Ax.5  Speed controlling
L2485  ; Ax.5  Speed-position switching l
L2486  ; Ax.5  Zero pass
L2489  ; Ax.5  Home position return reque
L2491  ; Ax.5  External signals FLS
L2492  ; Ax.5  External signals RLS
L2493  ; Ax.5  External signals STOP
L2494  ; Ax.5  External signals DOG/CHANG
L2495  ; Ax.5  Servo ready
L2496  ; Ax.5  Torque limiting
L2498  ; Ax.5  Virtual mode continuation
L2499  ; Ax.5 M-code outputting
L2500  ; Ax.6  Positioning start complete
L2502  ; Ax.6  In-position
L2503  ; Ax.6  Command in-position
L2504  ; Ax.6  Speed controlling
L2505  ; Ax.6  Speed-position switching l
L2506  ; Ax.6  Zero pass
L2509  ; Ax.6  Home position return reque
L2511  ; Ax.6  External signals FLS
L2512  ; Ax.6  External signals RLS
L2513  ; Ax.6  External signals STOP
L2514  ; Ax.6  External signals DOG/CHANG
L2515  ; Ax.6  Servo ready
L2516  ; Ax.6  Torque limiting
L2518  ; Ax.6  Virtual mode continuation
L2519  ; Ax.6 M-code outputting
L2520  ; Ax.7  Positioning start complete
L2521  ; Ax.7  Positioning complete
L2522  ; Ax.7  In-position
L2523  ; Ax.7  Command in-position
L2524  ; Ax.7  Speed controlling
L2525  ; Ax.7  Speed-position switching l
L2526  ; Ax.7  Zero pass
L2529  ; Ax.7  Home position return reque
L2531  ; Ax.7  External signals FLS
L2532  ; Ax.7  External signals RLS
L2533  ; Ax.7  External signals STOP
L2534  ; Ax.7  External signals DOG/CHANG
L2535  ; Ax.7  Servo ready
L2536  ; Ax.7  Torque limiting
L2538  ; Ax.7  Virtual mode continuation
L2539  ; Ax.7 M-code outputting
L2540  ; Ax.8  Positioning start complete
L2541  ; Ax.8  Positioning complete
L2542  ; Ax.8  In-position
L2543  ; Ax.8  Command in-position
L2544  ; Ax.8  Speed controlling
L2545  ; Ax.8  Speed-position switching l
L2546  ; Ax.8  Zero pass
L2547  ; Ax.8  Error detection
L2548  ; Ax.8  Servo error detection
L2549  ; Ax.8  Home position return reque
L2550  ; Ax.8  Home position return compl
L2551  ; Ax.8  External signals FLS
L2552  ; Ax.8  External signals RLS
L2553  ; Ax.8  External signals STOP
L2554  ; Ax.8  External signals DOG/CHANG
L2555  ; Ax.8  Servo ready
L2556  ; Ax.8  Torque limiting
L2558  ; Ax.8  Virtual mode continuation
L2559  ; Ax.8 M-code outputting
L3200  ; Ax.1  Stop command
L3201  ; Ax.1  Rapid stop command
L3202  ; Ax.1  Forward rotation JOG start
L3203  ; Ax.1  Reverse rotation JOG start
L3204  ; Ax.1  Complete signal OFF comman
L3205  ; Ax.1  Speed-position switching e
L3209  ; Ax.1  External stop input disabl
L3212  ; Ax.1  Feed current value update
L3213  ; Ax.1  Address clutch reference s
L3214  ; Ax.1  Cam reference position set
L3215  ; Ax.1  Servo OFF command
L3216  ; Ax.1  Gain changing command
L3218  ; Ax.1  Control loop changing comm
L3219  ; Ax.1 FIN signal
L3220  ; Ax.2  Stop command
L3221  ; Ax.2  Rapid stop command
L3222  ; Ax.2  Forward rotation JOG start
L3223  ; Ax.2  Reverse rotation JOG start
L3224  ; Ax.2  Complete signal OFF comman
L3225  ; Ax.2  Speed-position switching e
L3229  ; Ax.2  External stop input disabl
L3232  ; Ax.2  Feed current value update
L3233  ; Ax.2  Address clutch reference s
L3234  ; Ax.2  Cam reference position set
L3235  ; Ax.2  Servo OFF command
L3236  ; Ax.2  Gain changing command
L3238  ; Ax.2  Control loop changing comm
L3239  ; Ax.2 FIN signal
L3240  ; Ax.3  Stop command
L3241  ; Ax.3  Rapid stop command
L3242  ; Ax.3  Forward rotation JOG start
L3243  ; Ax.3  Reverse rotation JOG start
L3244  ; Ax.3  Complete signal OFF comman
L3245  ; Ax.3  Speed-position switching e
L3249  ; Ax.3  External stop input disabl
L3252  ; Ax.3  Feed current value update
L3253  ; Ax.3  Address clutch reference s
L3254  ; Ax.3  Cam reference position set
L3255  ; Ax.3  Servo OFF command
L3256  ; Ax.3  Gain changing command
L3258  ; Ax.3  Control loop changing comm
L3259  ; Ax.3 FIN signal
L3260  ; Ax.4  Stop command
L3261  ; Ax.4  Rapid stop command
L3262  ; Ax.4  Forward rotation JOG start
L3263  ; Ax.4  Reverse rotation JOG start
L3264  ; Ax.4  Complete signal OFF comman
L3265  ; Ax.4  Speed-position switching e
L3269  ; Ax.4  External stop input disabl
L3272  ; Ax.4  Feed current value update
L3273  ; Ax.4  Address clutch reference s
L3274  ; Ax.4  Cam reference position set
L3275  ; Ax.4  Servo OFF command
L3276  ; Ax.4  Gain changing command
L3278  ; Ax.4  Control loop changing comm
L3279  ; Ax.4 FIN signal
L3280  ; Ax.5  Stop command
L3281  ; Ax.5  Rapid stop command
L3282  ; Ax.5  Forward rotation JOG start
L3283  ; Ax.5  Reverse rotation JOG start
L3284  ; Ax.5  Complete signal OFF comman
L3285  ; Ax.5  Speed-position switching e
L3289  ; Ax.5  External stop input disabl
L3292  ; Ax.5  Feed current value update
L3293  ; Ax.5  Address clutch reference s
L3294  ; Ax.5  Cam reference position set
L3295  ; Ax.5  Servo OFF command
L3296  ; Ax.5  Gain changing command
L3298  ; Ax.5  Control loop changing comm
L3299  ; Ax.5 FIN signal
L3300  ; Ax.6  Stop command
L3301  ; Ax.6  Rapid stop command
L3302  ; Ax.6  Forward rotation JOG start
L3303  ; Ax.6  Reverse rotation JOG start
L3304  ; Ax.6  Complete signal OFF comman
L3305  ; Ax.6  Speed-position switching e
L3309  ; Ax.6  External stop input disabl
L3312  ; Ax.6  Feed current value update
L3313  ; Ax.6  Address clutch reference s
L3314  ; Ax.6  Cam reference position set
L3315  ; Ax.6  Servo OFF command
L3316  ; Ax.6  Gain changing command
L3318  ; Ax.6  Control loop changing comm
L3319  ; Ax.6 FIN signal
L3320  ; Ax.7  Stop command
L3321  ; Ax.7  Rapid stop command
L3322  ; Ax.7  Forward rotation JOG start
L3323  ; Ax.7  Reverse rotation JOG start
L3324  ; Ax.7  Complete signal OFF comman
L3325  ; Ax.7  Speed-position switching e
L3329  ; Ax.7  External stop input disabl
L3332  ; Ax.7  Feed current value update
L3333  ; Ax.7  Address clutch reference s
L3334  ; Ax.7  Cam reference position set
L3335  ; Ax.7  Servo OFF command
L3336  ; Ax.7  Gain changing command
L3338  ; Ax.7  Control loop changing comm
L3339  ; Ax.7 FIN signal
L3340  ; Ax.8  Stop command
L3341  ; Ax.8  Rapid stop command
L3342  ; Ax.8  Forward rotation JOG start
L3343  ; Ax.8  Reverse rotation JOG start
L3344  ; Ax.8  Complete signal OFF comman
L3345  ; Ax.8  Speed-position switching e
L3349  ; Ax.8  External stop input disabl
L3352  ; Ax.8  Feed current value update
L3353  ; Ax.8  Address clutch reference s
L3354  ; Ax.8  Cam reference position set
L3355  ; Ax.8  Servo OFF command
L3356  ; Ax.8  Gain changing command
L3358  ; Ax.8  Control loop changing comm
L3359  ; Ax.8 FIN signal
L4000  ; Virtual servo  Ax.1  Positioning
L4001  ; Virtual servo  Ax.1  Positioning
L4003  ; Virtual servo  Ax.1  Command in-
L4004  ; Virtual servo  Ax.1  Speed contr
L4007  ; Virtual servo  Ax.1  Error detec
L4019  ; Virtual servo  Ax.1  M-code outp
L4020  ; Virtual servo  Ax.2  Positioning
L4021  ; Virtual servo  Ax.2  Positioning
L4023  ; Virtual servo  Ax.2  Command in-
L4024  ; Virtual servo  Ax.2  Speed contr
L4027  ; Virtual servo  Ax.2  Error detec
L4039  ; Virtual servo  Ax.2  M-code outp
L4040  ; Virtual servo  Ax.3  Positioning
L4041  ; Virtual servo  Ax.3  Positioning
L4043  ; Virtual servo  Ax.3  Command in-
L4044  ; Virtual servo  Ax.3  Speed contr
L4047  ; Virtual servo  Ax.3  Error detec
L4059  ; Virtual servo  Ax.3  M-code outp
L4060  ; Virtual servo  Ax.4  Positioning
L4061  ; Virtual servo  Ax.4  Positioning
L4063  ; Virtual servo  Ax.4  Command in-
L4064  ; Virtual servo  Ax.4  Speed contr
L4067  ; Virtual servo  Ax.4  Error detec
L4079  ; Virtual servo  Ax.4  M-code outp
L4080  ; Virtual servo  Ax.5  Positioning
L4081  ; Virtual servo  Ax.5  Positioning
L4083  ; Virtual servo  Ax.5  Command in-
L4084  ; Virtual servo  Ax.5  Speed contr
L4087  ; Virtual servo  Ax.5  Error detec
L4099  ; Virtual servo  Ax.5  M-code outp
L4100  ; Virtual servo  Ax.6  Positioning
L4101  ; Virtual servo  Ax.6  Positioning
L4103  ; Virtual servo  Ax.6  Command in-
L4104  ; Virtual servo  Ax.6  Speed contr
L4107  ; Virtual servo  Ax.6  Error detec
L4119  ; Virtual servo  Ax.6  M-code outp
L4120  ; Virtual servo  Ax.7  Positioning
L4121  ; Virtual servo  Ax.7  Positioning
L4123  ; Virtual servo  Ax.7  Command in-
L4124  ; Virtual servo  Ax.7  Speed contr
L4127  ; Virtual servo  Ax.7  Error detec
L4139  ; Virtual servo  Ax.7  M-code outp
L4140  ; Virtual servo  Ax.8  Positioning
L4141  ; Virtual servo  Ax.8  Positioning
L4143  ; Virtual servo  Ax.8  Command in-
L4144  ; Virtual servo  Ax.8  Speed contr
L4147  ; Virtual servo  Ax.8  Error detec
L4159  ; Virtual servo  Ax.8  M-code outp
L4640  ; Sync. encoder  Ax.1  Error detec
L4641  ; Sync. encoder  Ax.1  External si
L4642  ; Sync. encoder  Ax.1  Virtual mod
L4644  ; Sync. encoder  Ax.2  Error detec
L4645  ; Sync. encoder  Ax.2  External si
L4646  ; Sync. encoder  Ax.2  Virtual mod
L4648  ; Sync. encoder  Ax.3  Error detec
L4649  ; Sync. encoder  Ax.3  External si
L4650  ; Sync. encoder  Ax.3  Virtual mod
L4652  ; Sync. encoder  Ax.4  Error detec
L4653  ; Sync. encoder  Ax.4  External si
L4654  ; Sync. encoder  Ax.4  Virtual mod
L4656  ; Sync. encoder  Ax.5  Error detec
L4657  ; Sync. encoder  Ax.5  External si
L4658  ; Sync. encoder  Ax.5  Virtual mod
L4660  ; Sync. encoder  Ax.6  Error detec
L4661  ; Sync. encoder  Ax.6  External si
L4662  ; Sync. encoder  Ax.6  Virtual mod
L4664  ; Sync. encoder  Ax.7  Error detec
L4665  ; Sync. encoder  Ax.7  External si
L4666  ; Sync. encoder  Ax.7  Virtual mod
L4668  ; Sync. encoder  Ax.8  Error detec
L4669  ; Sync. encoder  Ax.8  External si
L4670  ; Sync. encoder  Ax.8  Virtual mod
L4800  ; Virtual servo  Ax.1  Stop comman
L4801  ; Virtual servo  Ax.1  Rapid stop
L4802  ; Virtual servo  Ax.1  Forward rot
L4803  ; Virtual servo  Ax.1  Reverse rot
L4804  ; Virtual servo  Ax.1  Complete si
L4807  ; Virtual servo  Ax.1  Error reset
L4809  ; Virtual servo  Ax.1  External st
L4819  ; Virtual servo  Ax.1  FIN signal
L4820  ; Virtual servo  Ax.2  Stop comman
L4821  ; Virtual servo  Ax.2  Rapid stop
L4822  ; Virtual servo  Ax.2  Forward rot
L4823  ; Virtual servo  Ax.2  Reverse rot
L4824  ; Virtual servo  Ax.2  Complete si
L4827  ; Virtual servo  Ax.2  Error reset
L4829  ; Virtual servo  Ax.2  External st
L4839  ; Virtual servo  Ax.2  FIN signal
L4840  ; Virtual servo  Ax.3  Stop comman
L4841  ; Virtual servo  Ax.3  Rapid stop
L4842  ; Virtual servo  Ax.3  Forward rot
L4843  ; Virtual servo  Ax.3  Reverse rot
L4844  ; Virtual servo  Ax.3  Complete si
L4847  ; Virtual servo  Ax.3  Error reset
L4849  ; Virtual servo  Ax.3  External st
L4859  ; Virtual servo  Ax.3  FIN signal
L4860  ; Virtual servo  Ax.4  Stop comman
L4861  ; Virtual servo  Ax.4  Rapid stop
L4862  ; Virtual servo  Ax.4  Forward rot
L4863  ; Virtual servo  Ax.4  Reverse rot
L4864  ; Virtual servo  Ax.4  Complete si
L4867  ; Virtual servo  Ax.4  Error reset
L4869  ; Virtual servo  Ax.4  External st
L4879  ; Virtual servo  Ax.4  FIN signal
L4880  ; Virtual servo  Ax.5  Stop comman
L4881  ; Virtual servo  Ax.5  Rapid stop
L4882  ; Virtual servo  Ax.5  Forward rot
L4883  ; Virtual servo  Ax.5  Reverse rot
L4884  ; Virtual servo  Ax.5  Complete si
L4887  ; Virtual servo  Ax.5  Error reset
L4889  ; Virtual servo  Ax.5  External st
L4899  ; Virtual servo  Ax.5  FIN signal
L4900  ; Virtual servo  Ax.6  Stop comman
L4901  ; Virtual servo  Ax.6  Rapid stop
L4902  ; Virtual servo  Ax.6  Forward rot
L4903  ; Virtual servo  Ax.6  Reverse rot
L4904  ; Virtual servo  Ax.6  Complete si
L4907  ; Virtual servo  Ax.6  Error reset
L4909  ; Virtual servo  Ax.6  External st
L4919  ; Virtual servo  Ax.6  FIN signal
L4920  ; Virtual servo  Ax.7  Stop comman
L4921  ; Virtual servo  Ax.7  Rapid stop
L4922  ; Virtual servo  Ax.7  Forward rot
L4923  ; Virtual servo  Ax.7  Reverse rot
L4924  ; Virtual servo  Ax.7  Complete si
L4927  ; Virtual servo  Ax.7  Error reset
L4929  ; Virtual servo  Ax.7  External st
L4939  ; Virtual servo  Ax.7  FIN signal
L4940  ; Virtual servo  Ax.8  Stop comman
L4941  ; Virtual servo  Ax.8  Rapid stop
L4942  ; Virtual servo  Ax.8  Forward rot
L4943  ; Virtual servo  Ax.8  Reverse rot
L4944  ; Virtual servo  Ax.8  Complete si
L4947  ; Virtual servo  Ax.8  Error reset
L4949  ; Virtual servo  Ax.8  External st
L4959  ; Virtual servo  Ax.8  FIN signal
L5440  ; Sync. encoder  Ax.1  Error reset
L5444  ; Sync. encoder  Ax.2  Error reset
L5448  ; Sync. encoder  Ax.3  Error reset
L5452  ; Sync. encoder  Ax.4  Error reset
L5456  ; Sync. encoder  Ax.5  Error reset
L5460  ; Sync. encoder  Ax.6  Error reset
L5464  ; Sync. encoder  Ax.7  Error reset
L5468  ; Sync. encoder  Ax.8  Error reset
